_CFC_ (* Continuous Function Chart, elements in execution order *)
#0 INT_TO_TIME(SHU6_PV1_YA1_VREMYA_HODA)
#1 MUL(#0, 1000)
#2 stokeTime <= #1
#3 RT_PUSK:R_TRIG(CLK: SHU6_PV1_UST_RE_PUSK)
#4 TON_PCH_OTKL:TON(IN: SHU6_PV1_UST_RE_STOP, PT: T#1s)
#5 RT_PCH_OTKL:R_TRIG(CLK: #4.Q)
#6 RS_YA1_OPEN:RS(SET: #3.Q, RESET1: #5.Q)
#7 AND(NOT SHU6_PV1_MV1_DO3_VKL, NOT SHU6_PV1_YAMV1_DI8_M, SHU6_PV1_UST_RE_RABOTA)
#8 OR(SHU6_PV1_Z_MV1_AV, #7)
#9 SEL(SHU6_PV1_1YA1_DI5_A, eHVAC2PointActuatorMode_Close_OP, eHVAC2PointActuatorMode_Auto_BMS)
#10 SEL(#8, #9, eHVAC2PointActuatorMode_Close_OP)
#11 SHU6_PV1_1YA1_DO1_OTK <= #14.out 1
#12 OR(#14.out 4, #14.out 5)
#13 YA1_OTKAZ <= #12
#14 fb_HVACPAYa1:FB_HVAC2PointActuator(eHVACDataSecurityType_Idle, FALSE, TRUE, #6.Q1, #10, SHU6_PV1_KV1_DI6, SHU6_PV1_YA1_DI3_ZKR, SHU6_PV1_YA1_DI4_OTK, TRUE, SHU6_PV1_SB, enableLimitSwitch, stokeTime)
_END_CFC_
END_PROGRAM

(* POU IM/YA2_Upr, CFC *)
PROGRAM YA2_Upr
VAR
	RS_YA1_Open: RS;
	RT_Pusk: R_TRIG;
	RT_OSTANOV: R_TRIG;
	fb_HVACPA: FB_HVAC2PointActuator;

	stokeTime: TIME;
	enableLimitSwitch: BOOL := TRUE;
	FT_PCH_OTKL: R_TRIG;
	TON_PCH_OTKL: TON;
	ZADERJ_SHOD_YA1: TON;
	TON_YA1_Z_ZAM_TE6: TON;
END_VAR
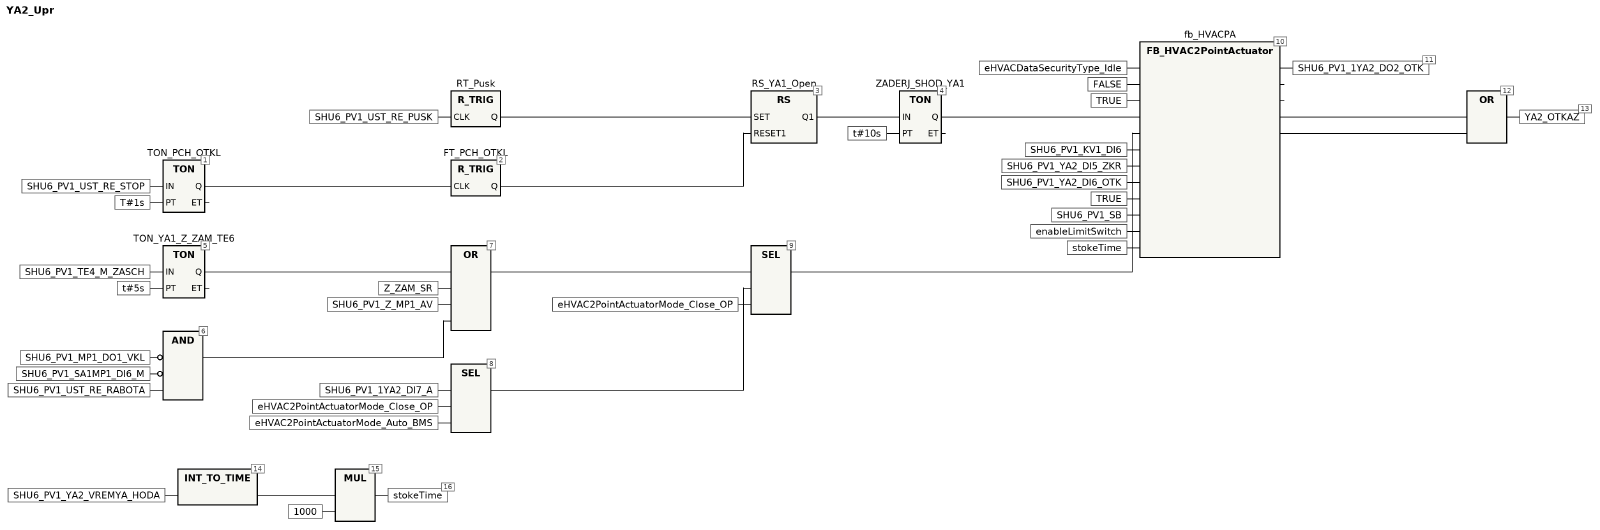
_CFC_ (* Continuous Function Chart, elements in execution order *)
#0 RT_Pusk:R_TRIG(CLK: SHU6_PV1_UST_RE_PUSK)
#1 TON_PCH_OTKL:TON(IN: SHU6_PV1_UST_RE_STOP, PT: T#1s)
#2 FT_PCH_OTKL:R_TRIG(CLK: #1.Q)
#3 RS_YA1_Open:RS(SET: #0.Q, RESET1: #2.Q)
#4 ZADERJ_SHOD_YA1:TON(IN: #3.Q1, PT: t#10s)
#5 TON_YA1_Z_ZAM_TE6:TON(IN: SHU6_PV1_TE4_M_ZASCH, PT: t#5s)
#6 AND(NOT SHU6_PV1_MP1_DO1_VKL, NOT SHU6_PV1_SA1MP1_DI6_M, SHU6_PV1_UST_RE_RABOTA)
#7 OR(#5.Q, Z_ZAM_SR, SHU6_PV1_Z_MP1_AV, #6)
#8 SEL(SHU6_PV1_1YA2_DI7_A, eHVAC2PointActuatorMode_Close_OP, eHVAC2PointActuatorMode_Auto_BMS)
#9 SEL(#7, #8, eHVAC2PointActuatorMode_Close_OP)
#10 fb_HVACPA:FB_HVAC2PointActuator(eHVACDataSecurityType_Idle, FALSE, TRUE, #4.Q, #9, SHU6_PV1_KV1_DI6, SHU6_PV1_YA2_DI5_ZKR, SHU6_PV1_YA2_DI6_OTK, TRUE, SHU6_PV1_SB, enableLimitSwitch, stokeTime)
#11 SHU6_PV1_1YA2_DO2_OTK <= #10.out 1
#12 OR(#10.out 4, #10.out 5)
#13 YA2_OTKAZ <= #12
#14 INT_TO_TIME(SHU6_PV1_YA2_VREMYA_HODA)
#15 MUL(#14, 1000)
#16 stokeTime <= #15
_END_CFC_
END_PROGRAM

(* POU IM/YA3_Upr, CFC *)
PROGRAM YA3_Upr
VAR
	YA3_PID: FB_HVACPIDCtrl;

	deadRange: REAL := 0.1;
	direction: BOOL;
	tTi: TIME;
	tTv: TIME;
	tTd: TIME;

	rYMin: REAL := 0;
	rYMax: REAL := 100;
	TON_SHU6_PV1_P1_DI5_RUN: TON;
	reg1: BOOL;
	reg2: BOOL;

	rwx: REAL;
	EPS1: REAL;
	EPS2: REAL;
END_VAR
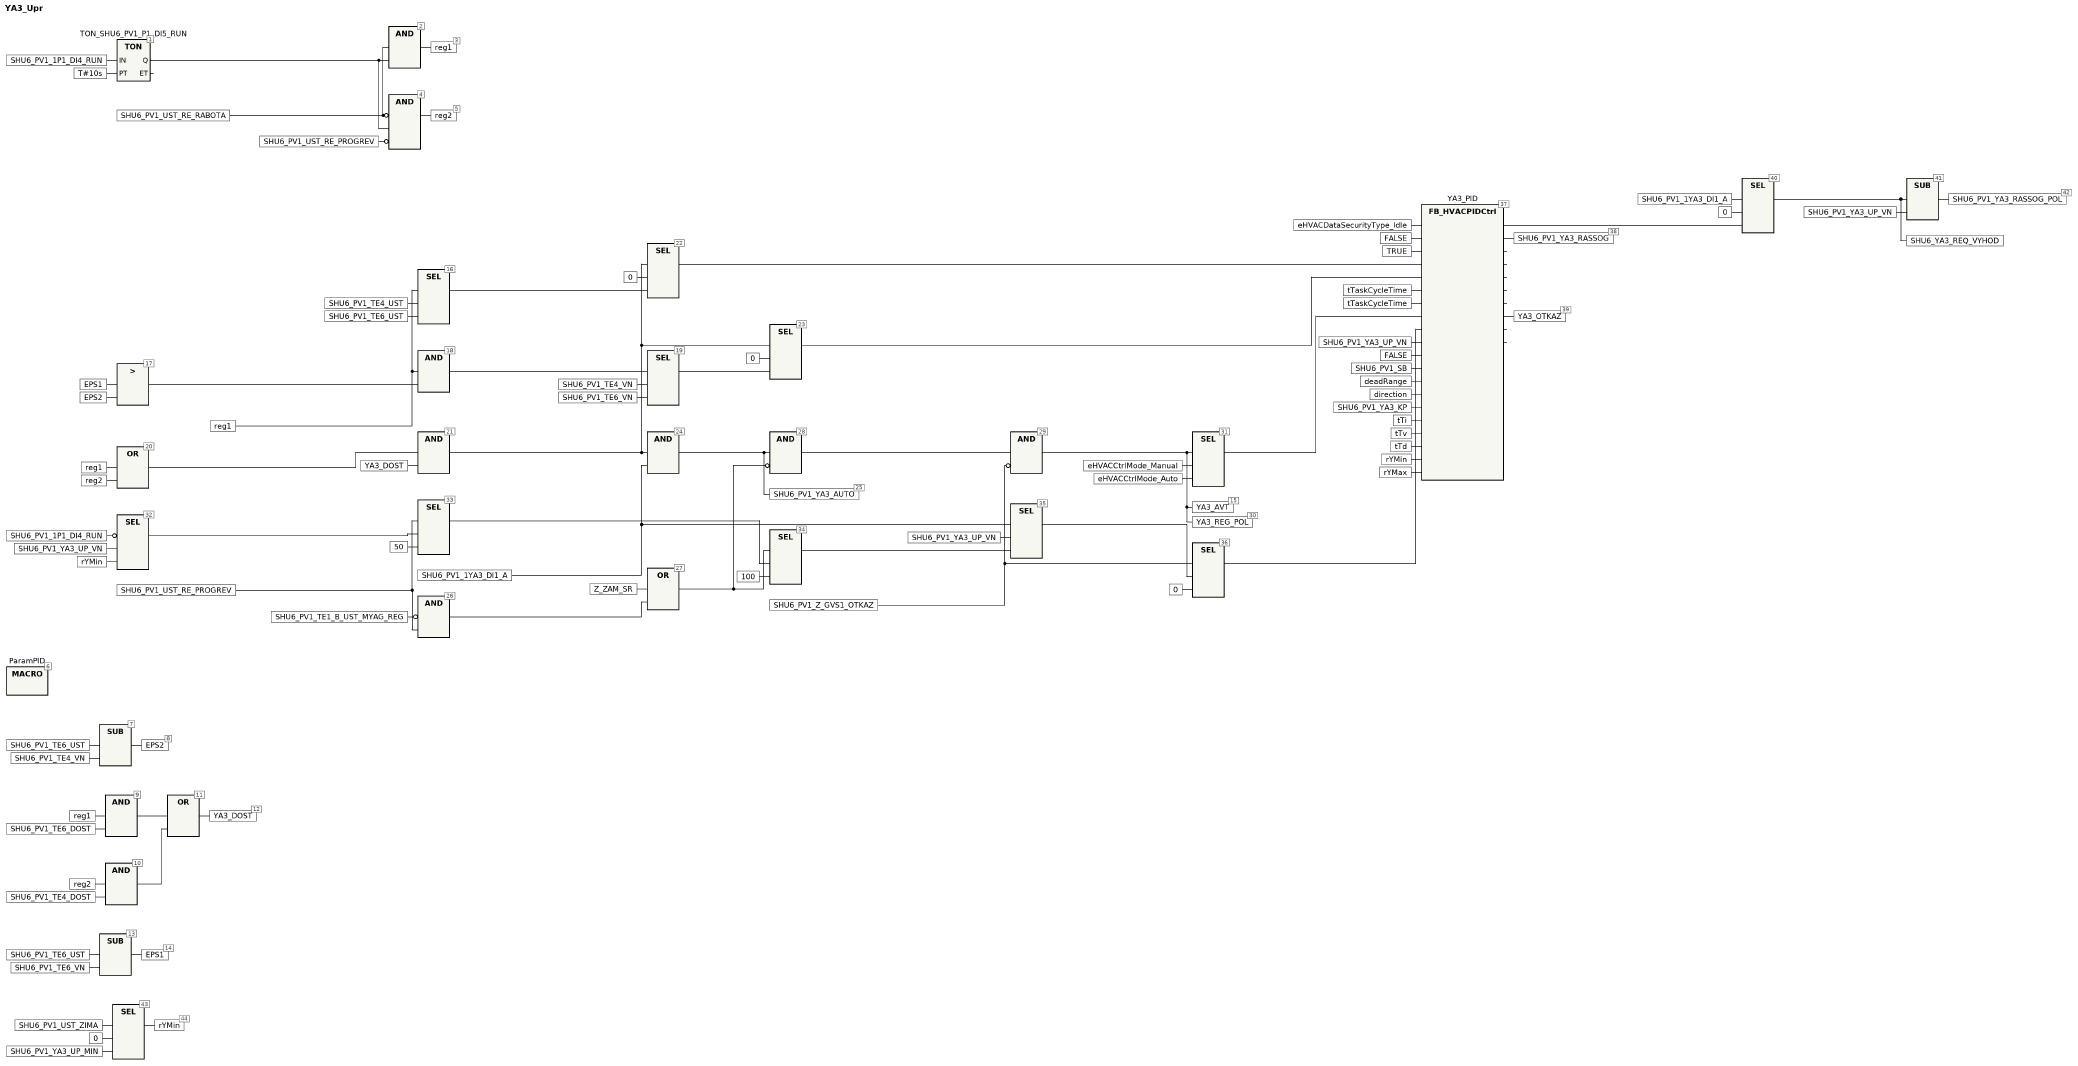
